FUNCTION_BLOCK FB_DigOutput_2
VAR_INPUT
	i_bStaOutput	: BOOL;
	i_stSettings 	: ST_DigOutputSettings;
	i_eCtrlMode		: E_CtrlMode;
	i_ref_eCtrlState : REFERENCE TO E_CtrlState;
END_VAR
VAR
//----------------------Outputs---------------------------//
	Q_bStaOutput AT %Q* : BOOL;
	
	// Force outputs (IO-test functions)
	s_fbForceCmdOutput : FB_ForceOutput;
	
//------------------------------------------------------//

//----------------------Properties---------------------------//
	{attribute 'hide'}
	s_bStaOutput			: BOOL;
	{attribute 'hide'}
	s_bStaOutputDelayed 	: BOOL;	
	{attribute 'hide'}
	s_bStaError			: BOOL;
	{attribute 'hide'}
	s_osrOn				: R_TRIG;
	{attribute 'hide'}
	s_osfOff		 	: F_TRIG;

//------------------------------------------------------//

//----------------------Variables---------------------------//
	s_bInitDone 	: BOOL;
	s_tonDelay 		: TON;
//------------------------------------------------------//

END_VAR


m_Main();

METHOD PRIVATE _m_Init : BOOL

s_bStaOutputDelayed := s_bStaOutput;

_m_Init := TRUE;
END_METHOD

METHOD PRIVATE _m_Outputs : BOOL
VAR_INST
	s_bCmdOutput : BOOL;
END_VAR

IF NOT i_stSettings.bCfgDelay THEN
	s_bCmdOutput := s_bStaOutput;
ELSE
	s_bCmdOutput := s_bStaOutputDelayed;
END_IF


IF __ISVALIDREF(i_ref_eCtrlState) THEN
	IF (i_eCtrlMode <> E_CtrlMode.IO) OR (i_ref_eCtrlState <> E_CtrlState.RUNNING) THEN
		s_fbForceCmdOutput.i_eForceValue := E_ForceValue.RELEASED; 	
	END_IF
END_IF
	
s_fbForceCmdOutput(
	i_ref_bCmdInput := s_bCmdOutput,
	i_ref_bCmdOutput := Q_bStaOutput);

_m_Outputs := TRUE;
END_METHOD

METHOD PUBLIC m_Main : BOOL

s_bStaOutput := i_bStaOutput;

IF NOT s_bInitDone THEN
	IF _m_Init() THEN
		s_bInitDone := TRUE;
	END_IF 
END_IF

s_osrOn(CLK := s_bStaOutput);
s_osfOff(CLK := s_bStaOutput);

s_tonDelay(IN := s_bStaOutput <> s_bStaOutputDelayed, PT := i_stSettings.tmOutputDelay);

IF s_bStaOutput AND s_tonDelay.Q THEN
	s_bStaOutputDelayed := TRUE;
END_IF

IF NOT s_bStaOutput AND s_tonDelay.Q THEN
	s_bStaOutputDelayed := FALSE;
END_IF

_m_Outputs();

m_Main := TRUE;
END_METHOD

{attribute 'monitoring':='call'}
PROPERTY PUBLIC p_bStaError : BOOL
GET
p_bStaError := s_bStaError;
END_GET
END_PROPERTY

{attribute 'monitoring':='call'}
PROPERTY PUBLIC p_bStaOutput : BOOL
GET
p_bStaOutput := s_bStaOutput;
END_GET
END_PROPERTY

{attribute 'monitoring':='call'}
PROPERTY PUBLIC p_bStaOutputDelayed : BOOL
GET
p_bStaOutputDelayed := s_bStaOutputDelayed;
END_GET
END_PROPERTY

{attribute 'monitoring':='call'}
PROPERTY PUBLIC p_osfOff : BOOL
GET
p_osfOff := s_osfOff.Q;
END_GET
END_PROPERTY

{attribute 'monitoring':='call'}
PROPERTY PUBLIC p_osrOn : BOOL
GET
p_osrOn := s_osrOn.Q;
END_GET
END_PROPERTY

END_FUNCTION_BLOCK

(* stored: Version 1.1.0.1, ProductVersion 3.1.4024.12
   POU FB_DigOutput_2: Id {f6926334-60a3-431a-8319-95017baa0ee2}, SpecialFunc None
   Method _m_Init: Id {58eaf209-c641-4c2f-b3df-64ebcea68410}
   Method _m_Outputs: Id {e570ab94-2a26-4b08-93d9-96af8fab708a}
   Method m_Main: Id {2dd33bfc-7121-4f83-aa70-6c1522573289}
   Property p_bStaError: Id {7a2eb779-abd4-40a3-9fc7-949ad97645b2}
   Get Get: Id {80d87ae8-eca1-4817-b904-fc6fac61aa99}
   Property p_bStaOutput: Id {cdc0ff34-12d0-4b48-b5e8-b09853bb5cc9}
   Get Get: Id {42e85b44-18f0-412a-9346-64d13e29ff2a}
   Property p_bStaOutputDelayed: Id {3637332a-480c-4238-8efd-ba968e49b075}
   Get Get: Id {68503e08-d1d6-43c3-9027-f0e9b82449cd}
   Property p_osfOff: Id {3b5a356d-bcf3-414b-9d28-f67f1ceb42ac}
   Get Get: Id {dcac5d8d-7ae8-4951-a311-58d0e8870f48}
   Property p_osrOn: Id {5e53c104-78f3-4605-a50c-a888c0276e40}
   Get Get: Id {b1ff90c4-6746-4d37-9bd2-d6308f16b98c} *)
